PROGRAM MAIN
VAR
	autoritenuta1	:	FB_Autoritenuta;
	autoritenuta2	:	FB_Autoritenuta;
END_VAR

autoritenuta1(start:= IO.bStart, stop:= IO.bStop , onoff=> IO.bHOn);

END_PROGRAM

(* stored: Version 1.1.0.1, ProductVersion 3.1.4024.12
   POU MAIN: Id {b76107a0-6f9d-49c7-b708-3794d1af63ed}, SpecialFunc None *)
